FUNCTION_BLOCK T_AddSameComponentTwiceShouldntAdd  EXTENDS T_UnitTestBase
VAR
  list : T_ComponentsCollection;
  newComponent : T_ComponentMock;
  actual : I_ComponentBase;
  expected : I_ComponentBase;
  result : BOOL;
END_VAR

list.AddComponent(newComponent);
result := NOT list.AddComponent(newComponent);

assertion.AssertEquals_BOOL(TRUE, result, 'result := NOT list.AddComponent(newComponent)');
TestFinished();

END_FUNCTION_BLOCK

(* stored: Version 1.1.0.1, ProductVersion 3.1.4024.12
   POU T_AddSameComponentTwiceShouldntAdd: Id {a93610e7-93f0-4e2f-8a19-8e4b314649ef}, SpecialFunc None *)
